TYPE ST_RecCtrl ://纠偏系统
STRUCT
    Cmd        :ST_RecCmd;
    Io            :ST_RecIo;
    Status      :ST_RecStatus;
END_STRUCT
END_TYPE

(* stored: Version 1.1.0.1, ProductVersion 3.1.4024.9
   DUT ST_RecCtrl: Id {962f8d4d-dc5f-45c6-8e4e-d0c353080fb3} *)
